{attribute 'qualified_only'}
{attribute 'strict'}
TYPE E_ComponentState :
(
	READY 	:= 0,
	BUSY	:= 1,
	DONE	:= 2
);
END_TYPE

(* stored: Version 1.1.0.1, ProductVersion 3.1.4024.15
   EnumerationTextList E_ComponentState: Id {1fad3293-1875-42d5-a862-59fd8ceefed0} *)
